// TIA Portal V17 export
// export: Created 2023-12-22T15:05:32.9936505Z, ExportSetting WithDefaults, DisplayName Totally Integrated Automation Portal, DisplayVersion V17, DisplayName TIA Portal Openness, DisplayVersion V17, DisplayName TIA Portal Version Control Interface, DisplayVersion V17, DisplayName STEP 7 Professional, DisplayVersion V17, DisplayName STEP 7 Safety, DisplayVersion V17, DisplayName WinCC Advanced, DisplayVersion V17
DATA_BLOCK "FB_DRV_Start_DB"   // DB100
VERSION : 0.1
// stored: AutoNumber false, DBAccessibleFromOPCUA true, InstanceOfName FB_DRV_Start, InstanceOfType FB
"FB_DRV_Start"
   // VAR
   //    last_01s : Int;
   //    last_05s : Int;
   //    last_1s : Int;
   //    last_5s : Int;
   //    last_10s : Int;
   //    last_30s : Int;
   //    last_1m : Int;
   //    last_5m : Int;
   //    last_10m : Int;
   //    last_30m : Int;
   //    last_1h : Int;
   //    last_1_day : Int;
   //    last_1_week : Int;
   //    last_1_month : Int;
   //    last_s1 : Int;
   //    last_s2 : Int;
   //    "1h_minutes" { S7_SetPoint := 'True'} : Int := 0;
   //    "1_day_hour" { S7_SetPoint := 'True'} : Int := 0;
   //    "1_day_minutes" { S7_SetPoint := 'True'} : Int := 0;
   //    "1_week_weekday" { S7_SetPoint := 'True'} : Int := 1;
   //    "1_week_hour" { S7_SetPoint := 'True'} : Int := 0;
   //    "1_week_minutes" { S7_SetPoint := 'True'} : Int := 0;
   //    "1_month_date" { S7_SetPoint := 'True'} : Int := 1;
   //    "1_month_hour" { S7_SetPoint := 'True'} : Int := 0;
   //    "1_month_minutes" { S7_SetPoint := 'True'} : Int := 0;
   //    s1_hour : Int;
   //    s1_minutes : Int;
   //    s2_hour : Int;
   //    s2_minutes : Int;
   //    pos : Array[0..15] of Bool;
   //    Error : Word;
   //    x { S7_SetPoint := 'True'} : "Protection";
   // END_VAR
BEGIN
   x.Stat[0..10] := FALSE;
   x.ADD_D := 7;
   x.Min_D := 7;
   x.Time_D.SP_D := 4;
   x.Time_D.SP_H := 0;
   x.Time_D.SP_M := 0;
   x.Time_D.SP_S := 0;
END_DATA_BLOCK
